PROGRAM MAIN
VAR
	_simpleContext : SimpleContext;
END_VAR

_simpleContext.Run();

END_PROGRAM

(* stored: Version 1.1.0.1, ProductVersion 3.1.4024.9
   POU MAIN: Id {ab5c28e5-92c3-456c-a9b3-a03f4b59ce35}, SpecialFunc None *)
